// TIA Portal V18 export
FUNCTION_BLOCK "Comms"   // FB22, LAD
TITLE = COMMS
{ S7_Optimized_Access := 'TRUE' }
// Written By Kristopher Gimenez March 3rd ,2023
// 
// This block and its associated DB are used to poll the profinet network for device status.
// stored: AutoNumber false, MemoryReserve 100, SetENOAutomatically false
   VAR
      DeviceLADDR : HW_IOSYSTEM := 273;   // 273 from Hardware identifier of PN network
      DeviceMode : UInt;
      DeviceReturn : Int;
      DeviceStates : Array[0..1023] of Bool;
      DeviceFault : Array[0..1023] of Bool;
      HpuPlcStatus : Bool;
      HpuPlcOnline : Bool;
      ConRIOStatus : Bool;
      ConRIOOnline : Bool;
      HpuHmiStatus : Bool;
      HpuHmiOnline : Bool;
      ConHmiStatus : Bool;
      ConHmiOnline : Bool;
      DHHmiStatus : Bool;
      DHHmiOnline : Bool;
      CouplerStatus : Bool;
      CouplerOnline : Bool;
      RemHearbeatOK : Bool;
      HBOn_TON { S7_SetPoint := 'True'} : TON_TIME;
      HeatbeatLost { S7_SetPoint := 'True'} : Bool;
      HBOff_TON { S7_SetPoint := 'True'} : TON_TIME;
      HBPosTrig : Bool;
      HBNegTrig : Bool;
   END_VAR
   VAR_TEMP
      RetVal : Int;
      TimeZone : Time;
      HmiTemp : Bool;
      BusyStatus : Bool;
   END_VAR
   VAR_TEMP   // added for the SCL form of the ladder/FBD networks
      _w1 : Bool;
      _w2 : Bool;
   END_VAR
BEGIN

REGION Network 2: Read the PLC local Time, HMI get the time.
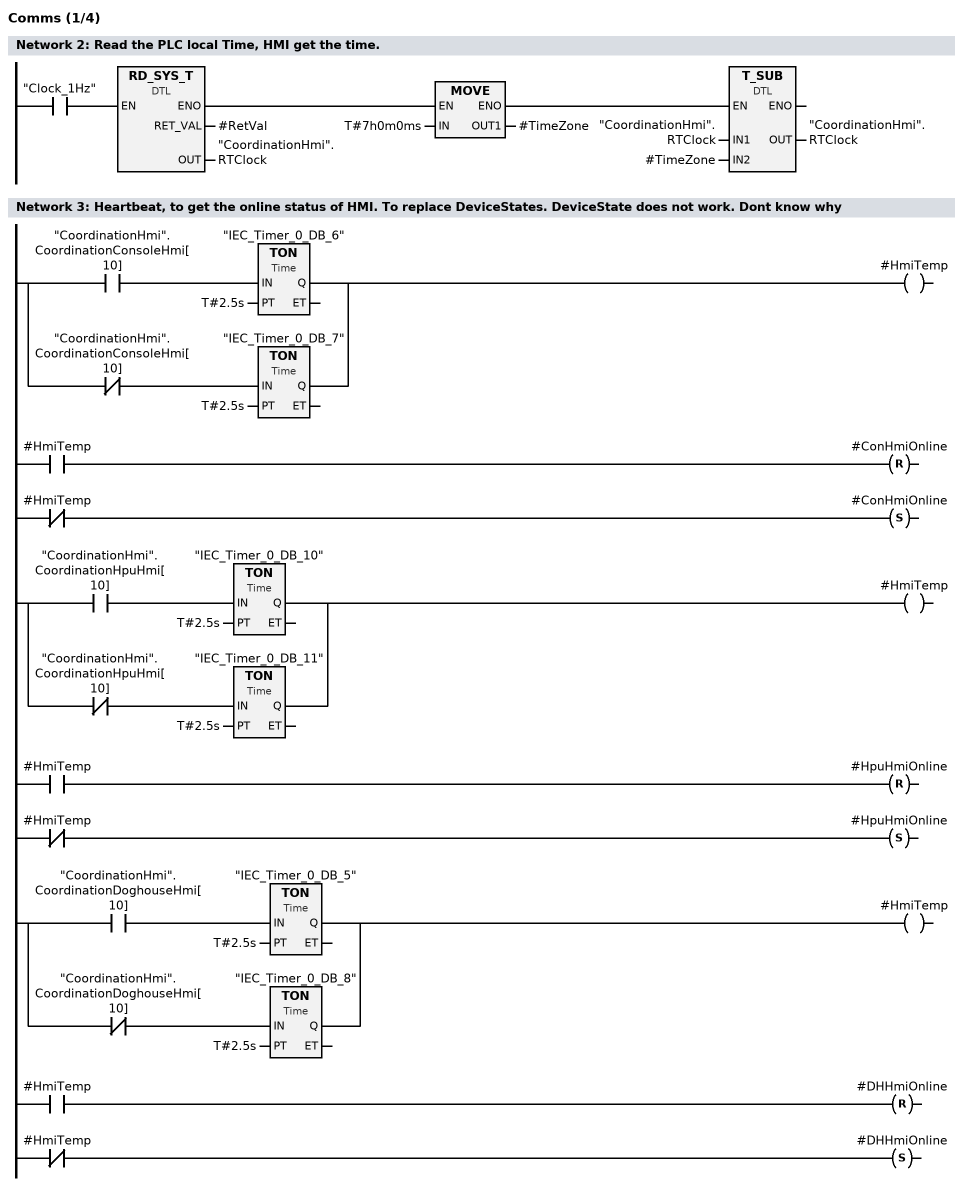
   RUNG wire#powerrail
      Contact( "Clock_1Hz" )
      { S7_Templates := "date_type := DTL" } RD_SYS_T(RET_VAL => #RetVal, OUT => "CoordinationHmi".RTClock)
      Move(in := T#7h0m0ms, out1 => #TimeZone)
      { S7_Templates := "[date_type := DTL, time_type := Time]" } T_SUB(IN1 := "CoordinationHmi".RTClock, IN2 := #TimeZone, OUT => "CoordinationHmi".RTClock)
   END_RUNG
   // the same network as SCL:
   #RetVal := RD_SYS_T(EN := "Clock_1Hz", OUT => "CoordinationHmi".RTClock, ENO => #_w1);
   IF #_w1 THEN
       #TimeZone := T#7h0m0ms;
       T_SUB(IN1 := "CoordinationHmi".RTClock, IN2 := #TimeZone, OUT => "CoordinationHmi".RTClock);
   END_IF;
END_REGION

REGION Network 3: Heartbeat, to get the online status of HMI. To replace DeviceStates. DeviceState does not work. Dont know why
   RUNG wire#powerrail
      Contact( "CoordinationHmi".CoordinationConsoleHmi[10] )
      { S7_Templates := "time_type := Time" } "IEC_Timer_0_DB_6".TON(pt := T#2.5s, et =>)
      wire#w1
      Coil( #HmiTemp )
   END_RUNG
   RUNG wire#powerrail
      I_Contact( "CoordinationHmi".CoordinationConsoleHmi[10] )
      { S7_Templates := "time_type := Time" } "IEC_Timer_0_DB_7".TON(pt := T#2.5s, et =>)
   END_RUNG wire#w1
   RUNG wire#powerrail
      Contact( #HmiTemp )
      R_Coil( #ConHmiOnline )
   END_RUNG
   RUNG wire#powerrail
      I_Contact( #HmiTemp )
      S_Coil( #ConHmiOnline )
   END_RUNG
   RUNG wire#powerrail
      Contact( "CoordinationHmi".CoordinationHpuHmi[10] )
      { S7_Templates := "time_type := Time" } "IEC_Timer_0_DB_10".TON(pt := T#2.5s, et =>)
      wire#w2
      Coil( #HmiTemp )
   END_RUNG
   RUNG wire#powerrail
      I_Contact( "CoordinationHmi".CoordinationHpuHmi[10] )
      { S7_Templates := "time_type := Time" } "IEC_Timer_0_DB_11".TON(pt := T#2.5s, et =>)
   END_RUNG wire#w2
   RUNG wire#powerrail
      Contact( #HmiTemp )
      R_Coil( #HpuHmiOnline )
   END_RUNG
   RUNG wire#powerrail
      I_Contact( #HmiTemp )
      S_Coil( #HpuHmiOnline )
   END_RUNG
   RUNG wire#powerrail
      Contact( "CoordinationHmi".CoordinationDoghouseHmi[10] )
      { S7_Templates := "time_type := Time" } "IEC_Timer_0_DB_5".TON(pt := T#2.5s, et =>)
      wire#w3
      Coil( #HmiTemp )
   END_RUNG
   RUNG wire#powerrail
      I_Contact( "CoordinationHmi".CoordinationDoghouseHmi[10] )
      { S7_Templates := "time_type := Time" } "IEC_Timer_0_DB_8".TON(pt := T#2.5s, et =>)
   END_RUNG wire#w3
   RUNG wire#powerrail
      Contact( #HmiTemp )
      R_Coil( #DHHmiOnline )
   END_RUNG
   RUNG wire#powerrail
      I_Contact( #HmiTemp )
      S_Coil( #DHHmiOnline )
   END_RUNG
   // the same network as SCL:
   "IEC_Timer_0_DB_6".TON(IN := "CoordinationHmi".CoordinationConsoleHmi[10], PT := T#2.5s);
   "IEC_Timer_0_DB_7".TON(IN := NOT "CoordinationHmi".CoordinationConsoleHmi[10], PT := T#2.5s);
   #HmiTemp := "IEC_Timer_0_DB_6".Q OR "IEC_Timer_0_DB_7".Q;
   IF #HmiTemp THEN #ConHmiOnline := FALSE; END_IF;
   IF NOT #HmiTemp THEN #ConHmiOnline := TRUE; END_IF;
   "IEC_Timer_0_DB_10".TON(IN := "CoordinationHmi".CoordinationHpuHmi[10], PT := T#2.5s);
   "IEC_Timer_0_DB_11".TON(IN := NOT "CoordinationHmi".CoordinationHpuHmi[10], PT := T#2.5s);
   #HmiTemp := "IEC_Timer_0_DB_10".Q OR "IEC_Timer_0_DB_11".Q;
   IF #HmiTemp THEN #HpuHmiOnline := FALSE; END_IF;
   IF NOT #HmiTemp THEN #HpuHmiOnline := TRUE; END_IF;
   "IEC_Timer_0_DB_5".TON(IN := "CoordinationHmi".CoordinationDoghouseHmi[10], PT := T#2.5s);
   "IEC_Timer_0_DB_8".TON(IN := NOT "CoordinationHmi".CoordinationDoghouseHmi[10], PT := T#2.5s);
   #HmiTemp := "IEC_Timer_0_DB_5".Q OR "IEC_Timer_0_DB_8".Q;
   IF #HmiTemp THEN #DHHmiOnline := FALSE; END_IF;
   IF NOT #HmiTemp THEN #DHHmiOnline := TRUE; END_IF;
END_REGION

REGION Network 4: Remote Console Heartbeat OK
   // Heartbeat is lost if state stays the same for the timeout time. Reset if Transition seen on heartbeat
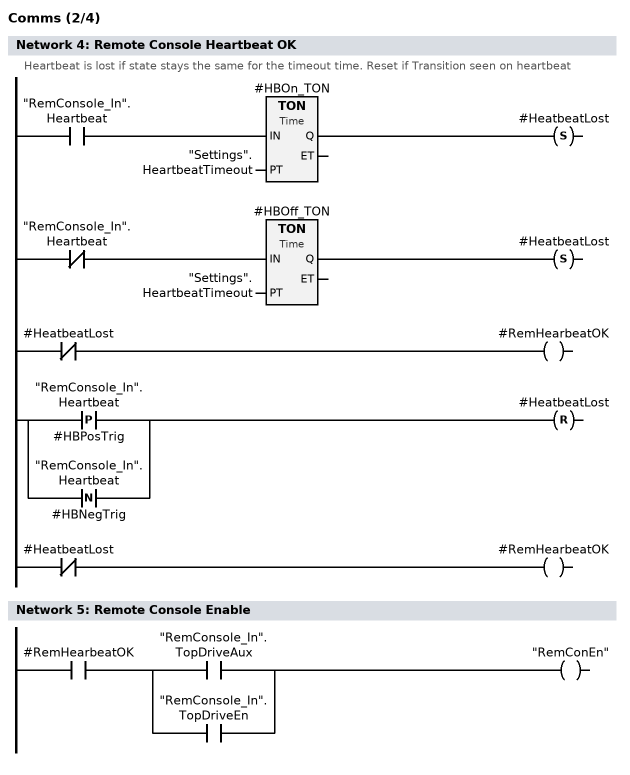
   RUNG wire#powerrail
      Contact( "RemConsole_In".Heartbeat )
      { S7_Templates := "time_type := Time" } #HBOn_TON.TON(pt := "Settings".HeartbeatTimeout, et =>)
      S_Coil( #HeatbeatLost )
   END_RUNG
   RUNG wire#powerrail
      I_Contact( "RemConsole_In".Heartbeat )
      { S7_Templates := "time_type := Time" } #HBOff_TON.TON(pt := "Settings".HeartbeatTimeout, et =>)
      S_Coil( #HeatbeatLost )
   END_RUNG
   RUNG wire#powerrail
      I_Contact( #HeatbeatLost )
      Coil( #RemHearbeatOK )
   END_RUNG
   RUNG wire#powerrail
      P_Contact(operand := "RemConsole_In".Heartbeat, bit := #HBPosTrig)
      wire#w1
      R_Coil( #HeatbeatLost )
   END_RUNG
   RUNG wire#powerrail
      N_Contact(operand := "RemConsole_In".Heartbeat, bit := #HBNegTrig)
   END_RUNG wire#w1
   RUNG wire#powerrail
      I_Contact( #HeatbeatLost )
      Coil( #RemHearbeatOK )
   END_RUNG
   // the same network as SCL:
   #HBOn_TON(IN := "RemConsole_In".Heartbeat, PT := "Settings".HeartbeatTimeout);   // TON
   IF #HBOn_TON.Q THEN #HeatbeatLost := TRUE; END_IF;
   #HBOff_TON(IN := NOT "RemConsole_In".Heartbeat, PT := "Settings".HeartbeatTimeout);   // TON
   IF #HBOff_TON.Q THEN #HeatbeatLost := TRUE; END_IF;
   #RemHearbeatOK := NOT #HeatbeatLost;
   #_w1 := "RemConsole_In".Heartbeat AND NOT #HBPosTrig;   // rising edge of "RemConsole_In".Heartbeat
   #HBPosTrig := "RemConsole_In".Heartbeat;
   #_w2 := NOT "RemConsole_In".Heartbeat AND #HBNegTrig;   // falling edge of "RemConsole_In".Heartbeat
   #HBNegTrig := "RemConsole_In".Heartbeat;
   IF #_w1 OR #_w2 THEN #HeatbeatLost := FALSE; END_IF;
   #RemHearbeatOK := NOT #HeatbeatLost;
END_REGION

REGION Network 5: Remote Console Enable
   RUNG wire#powerrail
      Contact( #RemHearbeatOK )
      wire#w1
      Contact( "RemConsole_In".TopDriveAux )
      wire#w2
      Coil( "RemConEn" )
   END_RUNG
   RUNG wire#w1
      Contact( "RemConsole_In".TopDriveEn )
   END_RUNG wire#w2
   // the same network as SCL:
   "RemConEn" := #RemHearbeatOK AND ("RemConsole_In".TopDriveAux OR "RemConsole_In".TopDriveEn);
END_REGION

REGION Network 6: Comms
   // Perform Device Exist check (mode 4) to see if device online
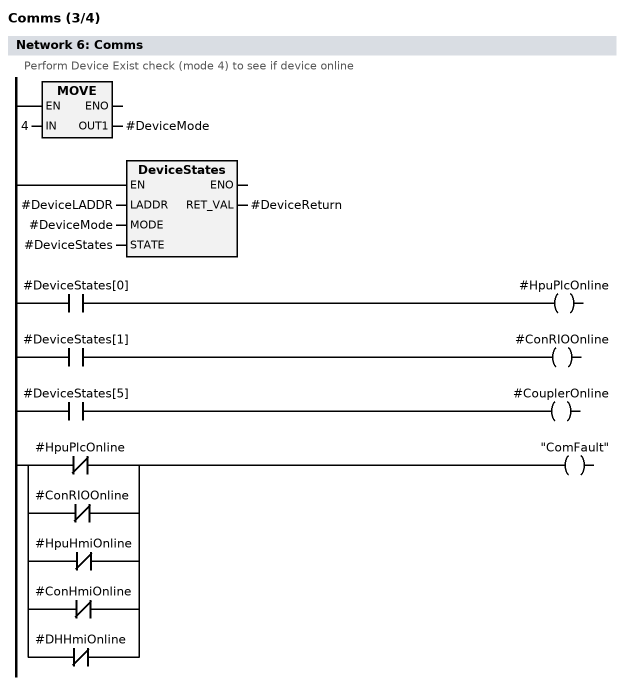
   RUNG wire#powerrail
      Move(in := 4, out1 => #DeviceMode)
   END_RUNG
   RUNG wire#powerrail
      DeviceStates(LADDR := #DeviceLADDR, MODE := #DeviceMode, STATE := #DeviceStates, Ret_Val => #DeviceReturn)
   END_RUNG
   RUNG wire#powerrail
      Contact( #DeviceStates[0] )
      Coil( #HpuPlcOnline )
   END_RUNG
   RUNG wire#powerrail
      Contact( #DeviceStates[1] )
      Coil( #ConRIOOnline )
   END_RUNG
   RUNG wire#powerrail
      Contact( #DeviceStates[5] )
      Coil( #CouplerOnline )
   END_RUNG
   RUNG wire#powerrail
      I_Contact( #HpuPlcOnline )
      wire#w1
      Coil( "ComFault" )
   END_RUNG
   RUNG wire#powerrail
      I_Contact( #ConRIOOnline )
   END_RUNG wire#w1
   RUNG wire#powerrail
      I_Contact( #HpuHmiOnline )
   END_RUNG wire#w1
   RUNG wire#powerrail
      I_Contact( #ConHmiOnline )
   END_RUNG wire#w1
   RUNG wire#powerrail
      I_Contact( #DHHmiOnline )
   END_RUNG wire#w1
   // the same network as SCL:
   #DeviceMode := 4;
   #DeviceReturn := DeviceStates(LADDR := #DeviceLADDR, MODE := #DeviceMode, STATE := #DeviceStates);
   #HpuPlcOnline := #DeviceStates[0];
   #ConRIOOnline := #DeviceStates[1];
   #CouplerOnline := #DeviceStates[5];
   "ComFault" := NOT #HpuPlcOnline OR NOT #ConRIOOnline OR NOT #HpuHmiOnline OR NOT #ConHmiOnline OR NOT #DHHmiOnline;
END_REGION

REGION Network 7: Fault State
   // Perform Device Fault check (mode 2) to see if device has fault. Set Status as Opposite. 1 = No Fault
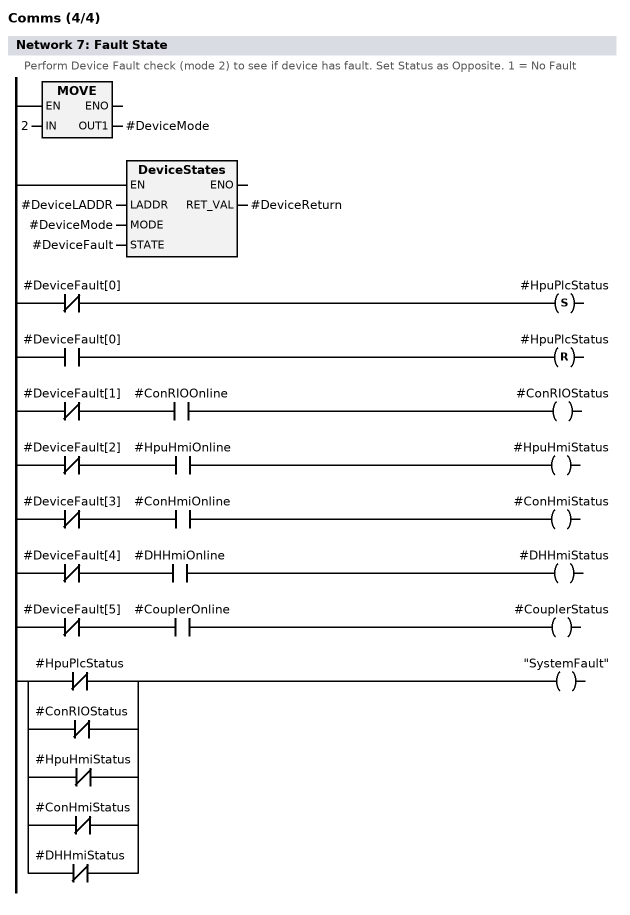
   RUNG wire#powerrail
      Move(in := 2, out1 => #DeviceMode)
   END_RUNG
   RUNG wire#powerrail
      DeviceStates(LADDR := #DeviceLADDR, MODE := #DeviceMode, STATE := #DeviceFault, Ret_Val => #DeviceReturn)
   END_RUNG
   RUNG wire#powerrail
      I_Contact( #DeviceFault[0] )
      S_Coil( #HpuPlcStatus )
   END_RUNG
   RUNG wire#powerrail
      Contact( #DeviceFault[0] )
      R_Coil( #HpuPlcStatus )
   END_RUNG
   RUNG wire#powerrail
      I_Contact( #DeviceFault[1] )
      Contact( #ConRIOOnline )
      Coil( #ConRIOStatus )
   END_RUNG
   RUNG wire#powerrail
      I_Contact( #DeviceFault[2] )
      Contact( #HpuHmiOnline )
      Coil( #HpuHmiStatus )
   END_RUNG
   RUNG wire#powerrail
      I_Contact( #DeviceFault[3] )
      Contact( #ConHmiOnline )
      Coil( #ConHmiStatus )
   END_RUNG
   RUNG wire#powerrail
      I_Contact( #DeviceFault[4] )
      Contact( #DHHmiOnline )
      Coil( #DHHmiStatus )
   END_RUNG
   RUNG wire#powerrail
      I_Contact( #DeviceFault[5] )
      Contact( #CouplerOnline )
      Coil( #CouplerStatus )
   END_RUNG
   RUNG wire#powerrail
      I_Contact( #HpuPlcStatus )
      wire#w1
      Coil( "SystemFault" )
   END_RUNG
   RUNG wire#powerrail
      I_Contact( #ConRIOStatus )
   END_RUNG wire#w1
   RUNG wire#powerrail
      I_Contact( #HpuHmiStatus )
   END_RUNG wire#w1
   RUNG wire#powerrail
      I_Contact( #ConHmiStatus )
   END_RUNG wire#w1
   RUNG wire#powerrail
      I_Contact( #DHHmiStatus )
   END_RUNG wire#w1
   // the same network as SCL:
   #DeviceMode := 2;
   #DeviceReturn := DeviceStates(LADDR := #DeviceLADDR, MODE := #DeviceMode, STATE := #DeviceFault);
   IF NOT #DeviceFault[0] THEN #HpuPlcStatus := TRUE; END_IF;
   IF #DeviceFault[0] THEN #HpuPlcStatus := FALSE; END_IF;
   #ConRIOStatus := NOT #DeviceFault[1] AND #ConRIOOnline;
   #HpuHmiStatus := NOT #DeviceFault[2] AND #HpuHmiOnline;
   #ConHmiStatus := NOT #DeviceFault[3] AND #ConHmiOnline;
   #DHHmiStatus := NOT #DeviceFault[4] AND #DHHmiOnline;
   #CouplerStatus := NOT #DeviceFault[5] AND #CouplerOnline;
   "SystemFault" := NOT #HpuPlcStatus OR NOT #ConRIOStatus OR NOT #HpuHmiStatus OR NOT #ConHmiStatus OR NOT #DHHmiStatus;
END_REGION
END_FUNCTION_BLOCK
